FUNCTION_BLOCK FB_PRECESS
VAR_INPUT
	ra				: LREAL;		// RA in degrees
	dec				: LREAL;		// Dec in degrees
	equinox1		: LREAL;		// epoch (Julian year) of the input coordinates
	equinox2		: LREAL;		// epoch (Julian year) of the output coordinates
END_VAR
VAR_OUTPUT
	ra_precessed	: LREAL;
	dec_precessed	: LREAL;
END_VAR
VAR
	ra_rad			: LREAL;		// RA in rad
	dec_rad			: LREAL;		// Dec in rad
	t				: LREAL;		// the elapsed time in Julian centuries since J2000 TT (days)
	EPS0, PSIA, OMEGAA, CHIA : LREAL;
	x, x2			: ARRAY[0..2] OF LREAL;
	rot				: ARRAY[0..2,0..2] OF LREAL;
	SA, CA, SB,CB,SC,CC,SD,CD: LREAL;
	step			: INT;			// 0: equinox1 -> J2000, 1: J2000 -> equinox2
	epoch			: LREAL;		// the non-J2000 epoch of the current step
END_VAR
VAR CONSTANT
	d2r 			: LREAL := PI/180.0;
	sec_to_rad 		: LREAL := d2r/3600.0;
END_VAR

(*
based on: NOVAS_F3.1.f -> SUBROUTINE PRECES
Kaplan, G., Bartlett, J., Monet, A., Bangert, J., & Puatua, W. (2011) User's Guide to NOVAS Version F3.1 (Washington, DC: USNO).

 THIS SUBROUTINE PRECESSES EQUATORIAL RECTANGULAR COORDINATES FROM
 ONE EPOCH TO ANOTHER.  THE COORDINATES ARE REFERRED TO THE MEAN
 DYNAMICAL EQUATOR AND EQUINOX OF THE TWO RESPECTIVE EPOCHS.  SEE
 EXPLANATORY SUPPLEMENT TO THE ASTRONOMICAL ALMANAC, PP. 103-104,
 AND CAPITAINE ET AL. (2003), ASTRONOMY AND ASTROPHYSICS 412,
 567-586.

 PRECES only rotates between J2000 and one other epoch, so a general
 equinox1 -> equinox2 is done in two steps via J2000. A step whose epoch
 is exactly 2000.0 is the identity and skipped.
*)

// deg 2 radian
ra_rad := ra*d2r;
dec_rad := dec*d2r;

x[0] := COS(dec_rad )*COS(ra_rad);
x[1] := COS(dec_rad )*SIN(ra_rad);
x[2] := SIN(dec_rad);


IF equinox1 <> equinox2 THEN
	FOR step := 0 TO 1 DO
		IF step = 0 THEN
			epoch := equinox1;
		ELSE
			epoch := equinox2;
		END_IF
		IF epoch <> 2000.0 THEN
			// t is the elapsed time in Julian centuries between J2000 and epoch
			t := 0.01*(epoch - 2000.0);
			EPS0 := sec_to_rad*	84381.406;
			PSIA := sec_to_rad*	( ( ( ( -    0.0000000951   * t
										+    0.000132851  ) * t
										-    0.00114045   ) * t
										-    1.0790069    ) * t
										+ 5038.481507     ) * t;
			OMEGAA := sec_to_rad*	( ( ( ( +    0.0000003337   * t
											-    0.000000467  ) * t
											-    0.00772503   ) * t
											+    0.0512623    ) * t
											-    0.025754     ) * t + EPS0;
			CHIA   := sec_to_rad*	( ( ( ( -    0.0000000560   * t
											+    0.000170663  ) * t
											-    0.00121197   ) * t
											-    2.3814292    ) * t
											+   10.556403     ) * t;
			SA := SIN(EPS0);
			CA := COS( EPS0 );
			SB := SIN( -PSIA );
			CB := COS( -PSIA );
			SC := SIN( -OMEGAA );
			CC := COS( -OMEGAA );
			SD := SIN( CHIA );
			CD := COS( CHIA );

			// COMPUTE ELEMENTS OF PRECESSION ROTATION MATRIX
			// EQUIVALENT TO R3(CHI_A)R1(-OMEGA_A)R3(-PSI_A)R1(EPSILON_0)
			rot[0,0] :=  CD * CB - SB * SD * CC; 	rot[0,1] := CD * SB * CA + SD * CC * CB * CA - SA * SD * SC; 	rot[0,2] := CD * SB * SA + SD * CC * CB * SA + CA * SD * SC;
			rot[1,0] := -SD * CB - SB * CD * CC; 	rot[1,1] := -SD * SB * CA + CD * CC * CB * CA - SA * CD * SC; 	rot[1,2] := -SD * SB * SA + CD * CC * CB * SA + CA * CD * SC;
			rot[2,0] := SB * SC;					rot[2,1] := -SC * CB * CA - SA * CC; 							rot[2,2] := -SC * CB * SA + CC * CA;

			// calculation as: Explanatory Supplement to the Astronomical Almanac (2013) p.220 eq.6.30
			//x2 := rot* x; //rotate to get output direction cosines
			IF step = 0 THEN
				// PERFORM ROTATION FROM EPOCH (equinox1) TO J2000.0
				x2[0] := rot[0,0]*x[0] + rot[1,0]*x[1] + rot[2,0]*x[2];
				x2[1] := rot[0,1]*x[0] + rot[1,1]*x[1] + rot[2,1]*x[2];
				x2[2] := rot[0,2]*x[0] + rot[1,2]*x[1] + rot[2,2]*x[2];
			ELSE
				// PERFORM ROTATION FROM J2000.0 TO EPOCH (equinox2)
				x2[0] := rot[0,0]*x[0] + rot[0,1]*x[1] + rot[0,2]*x[2];
				x2[1] := rot[1,0]*x[0] + rot[1,1]*x[1] + rot[1,2]*x[2];
				x2[2] := rot[2,0]*x[0] + rot[2,1]*x[1] + rot[2,2]*x[2];
			END_IF
			x[0] := x2[0];
			x[1] := x2[1];
			x[2] := x2[2];
		END_IF
	END_FOR
END_IF


ra_rad := atan2(x[1],x[0]);
dec_rad := ASIN(x[2]);

ra_precessed := ra_rad/d2r;
ra_precessed := MODABS(ra_precessed, 360.0);            //RA between 0 AND 360 degrees
dec_precessed := dec_rad/d2r;

END_FUNCTION_BLOCK

(* stored: Version 1.1.0.1, ProductVersion 3.1.4024.15
   POU FB_PRECESS: Id {879c3673-6766-4546-9283-3aa893f2e05f}, SpecialFunc None *)
